(* CODESYS project RepasoEjercicio1.project
   Title: RepasoEjercicio1
   Version: 0.0.0.0
   Author: bou

Project tree, tasks and I/O mapping:
  PLC_Cabecera_linea_ : TM241CE40R, Schneider Electric, order no. TM241CE40R, version 4.0.6.18
    application Application
      task MAST (cyclic, interval 20 ms, priority 15, watchdog 100 ms x 10) calls Control_Uno
      global variables GVL
      program Control_Uno [LD]
    DI : Digital Inputs, Schneider Electric, version 4.0.6.18
        input  idwDI_IDW0 : DWORD  // IDW0
        input  ibDI_IB1 : BYTE  // IB1
    DQ : Digital Outputs, Schneider Electric, version 4.0.6.18
        output qwDQ_QW0 : WORD  // QW0
        output qbDQ_QB1 : BYTE  // QB1
    Counters : Counters, Schneider Electric, version 4.0.6.18
    Pulse_Generators : Pulse Generators, Schneider Electric, version 4.0.6.18
    Cartridge_1 : Cartridge, Schneider Electric, version 4.0.6.18
    Cartridge_2 : Cartridge, Schneider Electric, version 4.0.6.18
    IO_Bus : IO bus - TM3, Schneider Electric, version 4.0.6.18
    COM_Bus : COM bus, Schneider Electric, version 4.0.6.18
    Ethernet_1 : Ethernet Network, Schneider Electric, version 4.0.6.18
        settings: IPAddress = [172, 16, 191, 108]; SubnetMask = [255, 255, 255, 0]; GatewayAddress = [172, 16, 191, 1]; WebServer = TRUE; FTP Server = TRUE; SoMachine Protocol = TRUE; Modbus Server = TRUE; NetManage Protocol = TRUE; SNMP protocol = TRUE; Enable Routing = FALSE; WebVisu protocol = TRUE; DHCP Server Active = FALSE
    Serial_Line_1 : Serial line, Schneider Electric, version 4.0.6.18
    Serial_Line_2 : Serial line, Schneider Electric, version 4.0.6.18
*)

// PLC_Cabecera_linea_/Application/GVL
VAR_GLOBAL
END_VAR

// PLC_Cabecera_linea_/Application/Control_Uno
PROGRAM Control_Uno
VAR
	Entrada_0 AT %IX0.0: BOOL;
	Entrada_1 AT %IX0.1: BOOL;
	Entrada_2 AT %IX0.2: BOOL;
	Entrada_3 AT %IX0.3: BOOL;
	Salida_0 AT %QX0.0: BOOL;
	Salida_1 AT %QX0.1: BOOL;
END_VAR

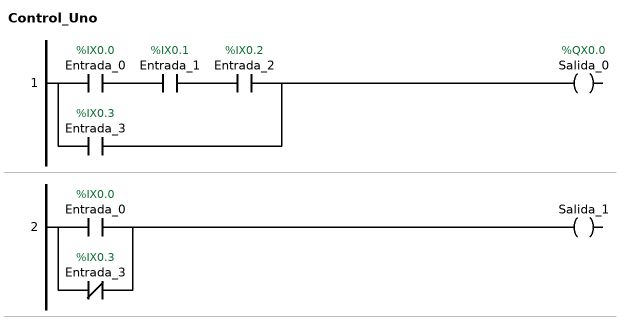
// NETWORK 1
//   Entrada_0: AT %IX0.0
//   Entrada_1: AT %IX0.1
//   Entrada_2: AT %IX0.2
//   Entrada_3: AT %IX0.3
//   Salida_0: AT %QX0.0
Salida_0 := Entrada_0 AND Entrada_1 AND Entrada_2 OR Entrada_3;

// NETWORK 2
//   Entrada_0: AT %IX0.0
//   Entrada_3: AT %IX0.3
Salida_1 := Entrada_0 OR NOT Entrada_3;

END_PROGRAM
